TYPE ST_Tank :
STRUCT
	nId : INT;
	fTemperature : REAL;
	fLevel : REAL;
	bTemperatureAlarm : BOOL;
	bLevelAlarm : BOOL;
END_STRUCT
END_TYPE

(* stored: Version 1.1.0.1, ProductVersion 3.1.4024.16
   DUT ST_Tank: Id {17a2f4de-6af3-4ef1-9617-ca64a6459c96} *)
